(* PLC project PLC_MarchaParo_POO_SinInterfaz, Beckhoff Automation GmbH TwinCAT PLC Control 3.5.20.60 *)
(* stored: creationDateTime 2026-08-25T11:45:00.0000000, modificationDateTime 2026-08-25T11:45:00.0000000 *)

FUNCTION_BLOCK FB_ControlMarchaParo
VAR
	_bSetaEmergenciaOk	AT %I*	: BOOL;
	_bPulsadorMarcha	AT %I*	: BOOL;
	_bPulsadorParo		AT %I*	: BOOL;
	_bPulsadorRearme	AT %I*	: BOOL;
	_bSalidaMotor		AT %Q*	: BOOL;
	
	_bEnMarcha					: BOOL;
	_bFalloSeguridad			: BOOL;
END_VAR

            
          

METHOD M_Cyclic
                  // Supervisión del canal de emergencia: corte inmediato y retención de fallo si el circuito se abre
IF NOT _bSetaEmergenciaOk THEN
    _bFalloSeguridad := TRUE;
    _bEnMarcha := FALSE;
END_IF

// Supervisión del pulsador de paro (contacto NC): detención inmediata al abrirse el contacto
IF NOT _bPulsadorParo THEN
    _bEnMarcha := FALSE;
END_IF

// Gestión del rearme físico: eliminación del flag de fallo si la seta física se encuentra en circuito cerrado
IF _bPulsadorRearme AND _bSetaEmergenciaOk THEN
    _bFalloSeguridad := FALSE;
END_IF

// Gestión del pulsador físico de marcha: activación del enclavamiento si se cumplen los requisitos de seguridad
IF _bPulsadorMarcha AND P_ListoParaMarcha THEN
    _bEnMarcha := TRUE;
END_IF

// Asignación continua del estado de marcha a la salida física
_bSalidaMotor := _bEnMarcha;
                
END_METHOD

METHOD M_Marcha : BOOL
                  // Activación de marcha por método: valida que la máquina esté lista y libre de fallos
IF P_ListoParaMarcha THEN
    _bEnMarcha := TRUE;
    M_Marcha := TRUE;
ELSE
    M_Marcha := FALSE;
END_IF
                
END_METHOD

METHOD M_Paro : BOOL
                  // Desconexión forzada del enclavamiento de marcha
_bEnMarcha := FALSE;
M_Paro := TRUE;
                
END_METHOD

METHOD M_Rearmar : BOOL
                  // Restablecimiento del estado de seguridad mediante comando si el canal de emergencia está cerrado
IF _bSetaEmergenciaOk THEN
    _bFalloSeguridad := FALSE;
    M_Rearmar := TRUE;
ELSE
    M_Rearmar := FALSE;
END_IF
                
END_METHOD

PROPERTY P_EmergenciaActiva : BOOL
GET
VAR
END_VAR
                    // Lectura del estado de emergencia: TRUE si hay fallo retenido o si la seta física está abierta
P_EmergenciaActiva := _bFalloSeguridad OR NOT _bSetaEmergenciaOk;
                  
END_GET
END_PROPERTY

PROPERTY P_EnMarcha : BOOL
GET
VAR
END_VAR
                    // Lectura del estado operativo: indica si el motor o actuador se encuentra actualmente activo
P_EnMarcha := _bEnMarcha;
                  
END_GET
END_PROPERTY

PROPERTY P_ListoParaMarcha : BOOL
GET
VAR
END_VAR
                    // Retorno de condición de disponibilidad: requiere ausencia de emergencias y paro en reposo
P_ListoParaMarcha := NOT P_EmergenciaActiva AND _bPulsadorParo;
                  
END_GET
END_PROPERTY
END_FUNCTION_BLOCK

PROGRAM MAIN
VAR
	fbMaquina			: FB_ControlMarchaParo;
	
	bCmdMarcha			: BOOL;
	bCmdParo			: BOOL;
	bCmdRearme			: BOOL;
	
	bEstadoEnMarcha		: BOOL;
	bEstadoEmergencia	: BOOL;
END_VAR

            // Ejecución periódica obligatoria de la lógica interna del bloque de control
fbMaquina.M_Cyclic();

// Procesamiento de comandos de control mediante métodos de la instancia
IF bCmdMarcha THEN
    fbMaquina.M_Marcha();
    bCmdMarcha := FALSE;
END_IF

IF bCmdParo THEN
    fbMaquina.M_Paro();
    bCmdParo := FALSE;
END_IF

IF bCmdRearme THEN
    fbMaquina.M_Rearmar();
    bCmdRearme := FALSE;
END_IF

// Lectura del estado operativo y de seguridad a través de las propiedades públicas
bEstadoEnMarcha := fbMaquina.P_EnMarcha;
bEstadoEmergencia := fbMaquina.P_EmergenciaActiva;
          
END_PROGRAM
